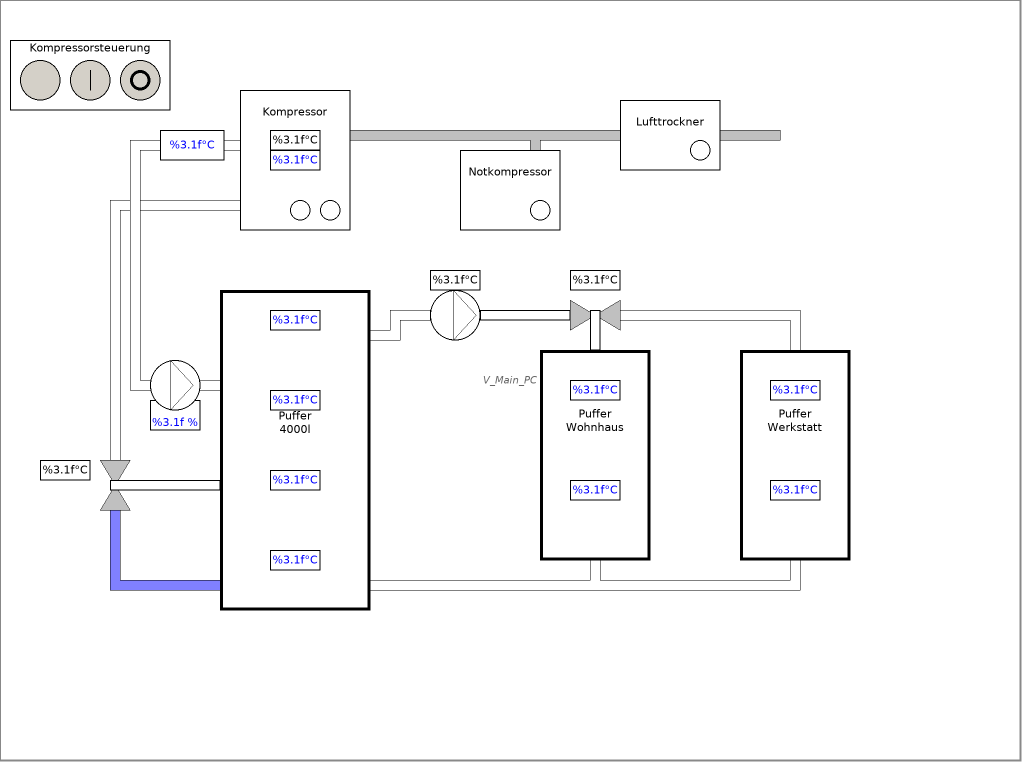
VISUALIZATION V_KomprWRG  // 1022x762
    Frame (0,0 1020x760)
        shows V_Main_PC()
    Polygon (330,130) (780,130) (780,140) (540,140) (540,150) (530,150) (530,140) (330,140)
    Polygon (570,300) (620,330) (620,300) (570,330) (570,320), colour toggle: PLC_PRG.fbKompressorSteuerung.QbVentilUmschWerkstatt
    Ellipse (430,290 50x50), colour toggle: PLC_PRG.fbKompressorSteuerung.QbUmwaelzpumpeWohnhaus
    Polygon (453,290) (476,315) (453,340) (453,327)
    Rectangle (480,310 90x10), colour toggle: PLC_PRG.fbKompressorSteuerung.QbUmwaelzpumpeWohnhaus
    Rectangle (590,310 10x40), colour toggle: PLC_PRG.fbKompressorSteuerung.QbVentilUmschWerkstatt
    Polygon (620,310) (800,310) (800,350) (790,350) (790,320) (620,320), colour toggle: PLC_PRG.fbKompressorSteuerung.QbUmwaelzpumpeWohnhaus and not PLC_PRG.fbKompressorSteuerung.QbVentilUmschWerkstatt
    Polygon (370,580) (390,580) (410,580) (590,580) (590,560) (600,560) (600,580) (790,580) (790,560) (800,560) (800,580) (800,590) (400,590) (390,590) (370,590), colour toggle: PLC_PRG.fbKompressorSteuerung.QbUmwaelzpumpeWohnhaus
    Rectangle (150,400 50x30), "%3.1f %", text variable: PLC_PRG.fbKompressorSteuerung.fbAnalogOutUmwaelzpumpeWRG.INrValue * 100
    Rectangle (240,90 110x140), "Kompressor"
    Rectangle (460,150 100x80), "Notkompressor"
    Rectangle (620,100 100x70), "Lufttrockner"
    Ellipse (690,140 20x20), colour toggle: PLC_PRG.fbKompressorSteuerung.QbLufttrockner
    Ellipse (530,200 20x20), colour toggle: PLC_PRG.fbKompressorSteuerung.QbNotKompressor
    Ellipse (320,200 20x20), colour toggle: PLC_PRG.fbKompressorSteuerung.QbKompressor
    Ellipse (290,200 20x20), tooltip "Störung", colour toggle: PLC_PRG.fbKompressorSteuerung.IbStoerung
    Polygon (100,510) (130,460) (100,460) (130,510) (130,510), colour toggle: PLC_PRG.fbKompressorSteuerung.QbVentilSchnellauflWRG
    Rectangle (110,480 110x10), colour toggle: PLC_PRG.fbKompressorSteuerung.QbVentilSchnellauflWRG
    Polygon (110,510) (110,590) (220,590) (220,580) (120,580) (120,510), colour toggle: PLC_PRG.fbKompressorSteuerung.QbVentilSchnellauflWRG
    Polygon (240,210) (120,210) (120,460) (110,460) (110,200) (240,200), colour toggle: PLC_PRG.fbKompressorSteuerung.QbUmwaelzpumpeWRG
    Polygon (240,140) (130,140) (130,390) (220,390) (220,380) (140,380) (140,150) (240,150), colour toggle: PLC_PRG.fbKompressorSteuerung.QbUmwaelzpumpeWRG
    Ellipse (150,360 50x50), colour toggle: PLC_PRG.fbKompressorSteuerung.QbUmwaelzpumpeWRG
    Polygon (170,360) (193,385) (170,410) (170,397)
    Rectangle (160,130 64x30), "%3.1f°C", text variable: gfbTemp31_KomprWRG_Ruecklauf.OUTrValue
    Rectangle (270,150 50x20), "%3.1f°C", text variable: gfbTemp32_KomprWRG_Vorlauf.OUTrValue
    Rectangle (40,460 50x20), "%3.1f°C", tooltip "Temperatur, Umschaltung Schnellaufladung", text variable: PLC_PRG.fbKompressorSteuerung.VrKomprWRG_TempSchnellaufl
        OnMouseClick: write the text variable via Default, min 20, max 70
    Rectangle (270,130 50x20), "%3.1f°C", tooltip "Solltemperatur Vorlauf", text variable: PLC_PRG.fbKompressorSteuerung.VrKomprWRG_TempVorlaufSollwert
        OnMouseClick: write the text variable via Default, min 20, max 80
    Rectangle (430,270 50x20), "%3.1f°C", tooltip "Temperatur, Umschaltung zum Wohnhaus", text variable: PLC_PRG.fbKompressorSteuerung.VrKomprWRG_TempUmschaltZurWohnh
        OnMouseClick: write the text variable via Default, min 20, max 70
    Rectangle (570,270 50x20), "%3.1f°C", tooltip "Temperatur, Umschaltung zur Werkstatt", text variable: PLC_PRG.fbKompressorSteuerung.VrKomprWRG_TempUmschaltZurWerkst
        OnMouseClick: write the text variable via Default, min 20, max 70
    Polygon (430,310) (430,320) (400,320) (400,340) (370,340) (370,330) (390,330) (390,310), colour toggle: PLC_PRG.fbKompressorSteuerung.QbUmwaelzpumpeWohnhaus
    Rectangle (10,40 160x70), "Kompressorsteuerung"
    Ellipse (20,60 40x40), tooltip "Störung", colour toggle: PLC_PRG.fbKompressorSteuerung.QbLMStatus
    Ellipse (70,60 40x40), tooltip "Störung", colour toggle: PLC_PRG.fbKompressorSteuerung.VbStart
        tap PLC_PRG.fbKompressorSteuerung.VbStart
    Ellipse (120,60 40x40), tooltip "Störung", colour toggle: PLC_PRG.fbKompressorSteuerung.VbStop
        tap PLC_PRG.fbKompressorSteuerung.VbStop
    RoundedRectangle (222,520 146x88), colour variable: gfbTemp14_Puffer4000_unten.VdiColourOfTemperature
    Ellipse (130,70 20x20)
    Line (90,70) (90,90)
    RoundedRectangle (222,440 146x95), colour variable: gfbTemp13_Puffer4000_mitte.VdiColourOfTemperature
    RoundedRectangle (222,360 146x95), colour variable: gfbTemp12_Puffer4000_oben.VdiColourOfTemperature
    RoundedRectangle (222,292 146x85), colour variable: gfbTemp11_Puffer4000_Brauchw.VdiColourOfTemperature
    RoundedRectangle (220,290 150x320), "Puffer 4000l"
    Rectangle (270,390 50x20), "%3.1f°C", text variable: gfbTemp12_Puffer4000_oben.OUTrValue
    Rectangle (270,470 50x20), "%3.1f°C", text variable: gfbTemp13_Puffer4000_mitte.OUTrValue
    Rectangle (270,550 50x20), "%3.1f°C", text variable: gfbTemp14_Puffer4000_unten.OUTrValue
    Rectangle (270,310 50x20), "%3.1f°C", text variable: gfbTemp11_Puffer4000_Brauchw.OUTrValue
    RoundedRectangle (742,450 106x108), colour variable: gfbTemp24_PufferWerkst_unten.VdiColourOfTemperature
    RoundedRectangle (742,352 106x110), colour variable: gfbTemp23_PufferWerkst_oben.VdiColourOfTemperature
    RoundedRectangle (740,350 110x210), "Puffer Werkstatt"
    Rectangle (770,480 50x20), "%3.1f°C", text variable: gfbTemp24_PufferWerkst_unten.OUTrValue
    Rectangle (770,380 50x20), "%3.1f°C", text variable: gfbTemp23_PufferWerkst_oben.OUTrValue
    RoundedRectangle (542,448 106x108), colour variable: gfbTemp22_PufferWohnh_unten.VdiColourOfTemperature
    RoundedRectangle (542,352 106x110), colour variable: gfbTemp21_PufferWohnh_oben.VdiColourOfTemperature
    Rectangle (570,480 50x20), "%3.1f°C", text variable: gfbTemp22_PufferWohnh_unten.OUTrValue
    Rectangle (570,380 50x20), "%3.1f°C", text variable: gfbTemp21_PufferWohnh_oben.OUTrValue
    RoundedRectangle (540,350 110x210), "Puffer Wohnhaus"
END_VISUALIZATION

(* stored: Version 1.1.0.1, ProductVersion 3.1.4018.5
   Visu V_KomprWRG: Id {1d64e77e-0ed0-4e1d-a4c2-aac45d1b02f7} *)
